PROGRAM OP90_MASTER3_IO
VAR
    OP90_MAS3_PORT1_BYTE1_DI_MODULE_1 AT %I* : BYTE;
	OP90_MAS3_PORT1_BYTE2_DI_MODULE_1 AT %I* : BYTE;
	OP90_MAS3_PORT2_BYTE1_DI_MODULE_2 AT %I* : BYTE;
	OP90_MAS3_PORT2_BYTE2_DI_MODULE_2 AT %I* : BYTE;
	OP90_MAS3_PORT3_BYTE1_DI_MODULE_3 AT %I* : BYTE;
	OP90_MAS3_PORT3_BYTE2_DI_MODULE_3 AT %I* : BYTE;
	
	OP90_MAS3_PORT5_BYTE1_DO_MODULE_1 AT %Q* : BYTE;
	OP90_MAS3_PORT5_BYTE2_DO_MODULE_1 AT %Q* : BYTE;
	OP90_MAS3_PORT5_BYTE3_DO_MODULE_1 AT %Q* : BYTE;
	OP90_MAS3_PORT6_BYTE1_DO_MODULE_2 AT %Q* : BYTE;
	OP90_MAS3_PORT6_BYTE2_DO_MODULE_2 AT %Q* : BYTE;
	OP90_MAS3_PORT7_BYTE1_DO_MODULE_3 AT %Q* : BYTE; 
	OP90_MAS3_PORT7_BYTE2_DO_MODULE_3 AT %Q* : BYTE;
	OP90_MAS3_PORT7_BYTE3_DO_MODULE_3 AT %Q* : BYTE;
	
	

	BYTE_AS_BIT_0: BYTE_AS_BIT;
	BYTE_AS_BIT_1: BYTE_AS_BIT;
	BYTE_AS_BIT_2: BYTE_AS_BIT;
	BYTE_AS_BIT_3: BYTE_AS_BIT;
	BYTE_AS_BIT_4: BYTE_AS_BIT;
	BYTE_AS_BIT_5: BYTE_AS_BIT;
	
	
	
	BIT_AS_BYTE_0: BIT_AS_BYTE;
	BIT_AS_BYTE_1: BIT_AS_BYTE;
	BIT_AS_BYTE_2: BIT_AS_BYTE;
	BIT_AS_BYTE_3: BIT_AS_BYTE;
	BIT_AS_BYTE_4: BIT_AS_BYTE;
	BIT_AS_BYTE_5: BIT_AS_BYTE;
	BIT_AS_BYTE_6: BIT_AS_BYTE;
	BIT_AS_BYTE_7: BIT_AS_BYTE;
		
END_VAR

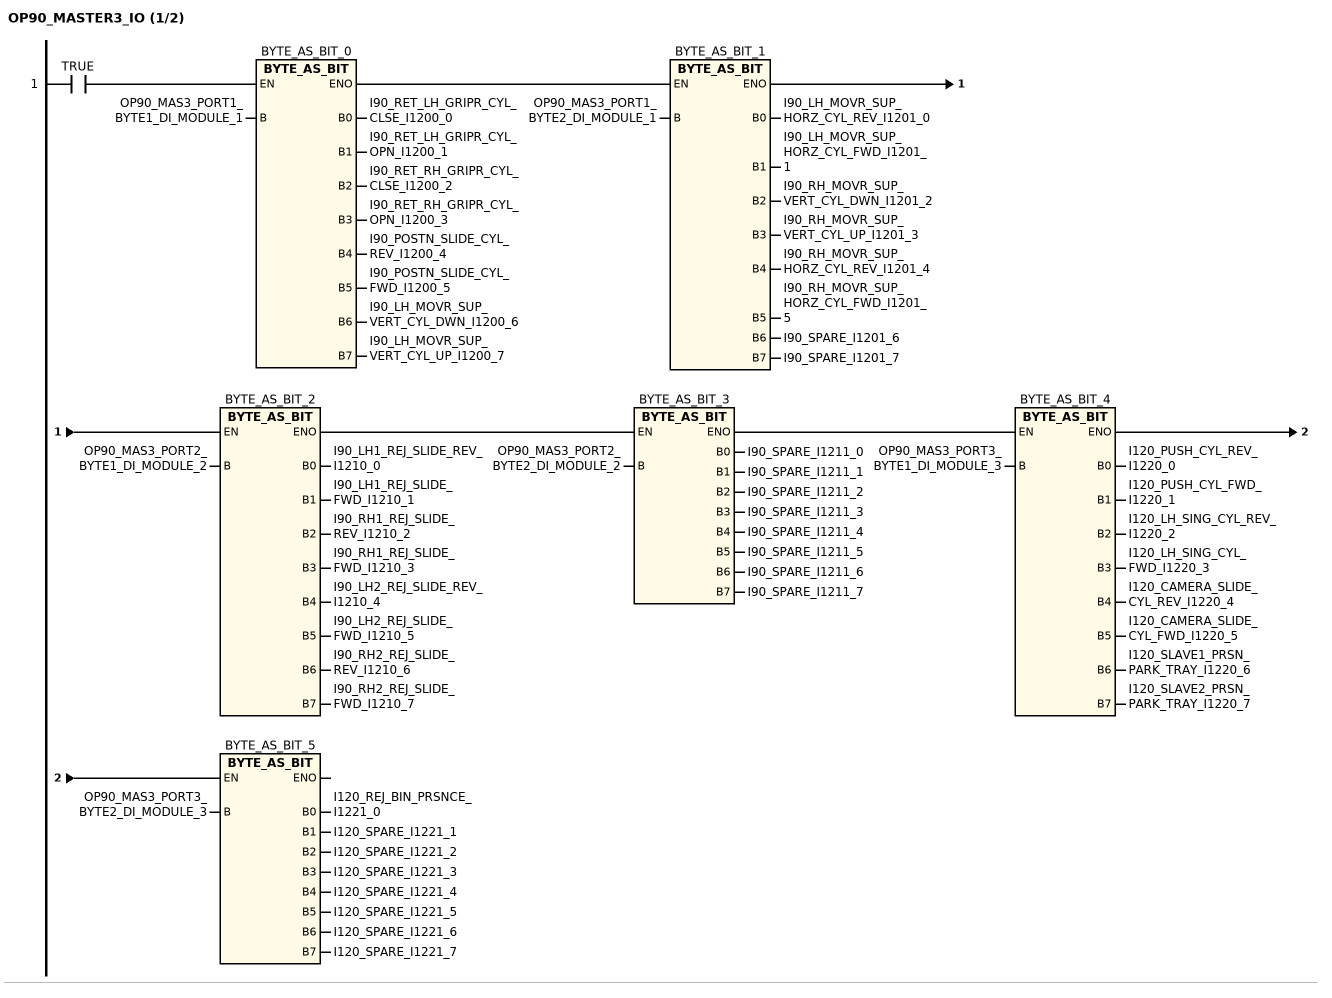
// NETWORK 1
BYTE_AS_BIT_0(
    B := OP90_MAS3_PORT1_BYTE1_DI_MODULE_1,
    B0 => I90_RET_LH_GRIPR_CYL_CLSE_I1200_0,
    B1 => I90_RET_LH_GRIPR_CYL_OPN_I1200_1,
    B2 => I90_RET_RH_GRIPR_CYL_CLSE_I1200_2,
    B3 => I90_RET_RH_GRIPR_CYL_OPN_I1200_3,
    B4 => I90_POSTN_SLIDE_CYL_REV_I1200_4,
    B5 => I90_POSTN_SLIDE_CYL_FWD_I1200_5,
    B6 => I90_LH_MOVR_SUP_VERT_CYL_DWN_I1200_6,
    B7 => I90_LH_MOVR_SUP_VERT_CYL_UP_I1200_7); // BYTE_AS_BIT
BYTE_AS_BIT_1(
    B := OP90_MAS3_PORT1_BYTE2_DI_MODULE_1,
    B0 => I90_LH_MOVR_SUP_HORZ_CYL_REV_I1201_0,
    B1 => I90_LH_MOVR_SUP_HORZ_CYL_FWD_I1201_1,
    B2 => I90_RH_MOVR_SUP_VERT_CYL_DWN_I1201_2,
    B3 => I90_RH_MOVR_SUP_VERT_CYL_UP_I1201_3,
    B4 => I90_RH_MOVR_SUP_HORZ_CYL_REV_I1201_4,
    B5 => I90_RH_MOVR_SUP_HORZ_CYL_FWD_I1201_5,
    B6 => I90_SPARE_I1201_6,
    B7 => I90_SPARE_I1201_7); // BYTE_AS_BIT
BYTE_AS_BIT_2(
    B := OP90_MAS3_PORT2_BYTE1_DI_MODULE_2,
    B0 => I90_LH1_REJ_SLIDE_REV_I1210_0,
    B1 => I90_LH1_REJ_SLIDE_FWD_I1210_1,
    B2 => I90_RH1_REJ_SLIDE_REV_I1210_2,
    B3 => I90_RH1_REJ_SLIDE_FWD_I1210_3,
    B4 => I90_LH2_REJ_SLIDE_REV_I1210_4,
    B5 => I90_LH2_REJ_SLIDE_FWD_I1210_5,
    B6 => I90_RH2_REJ_SLIDE_REV_I1210_6,
    B7 => I90_RH2_REJ_SLIDE_FWD_I1210_7); // BYTE_AS_BIT
BYTE_AS_BIT_3(
    B := OP90_MAS3_PORT2_BYTE2_DI_MODULE_2,
    B0 => I90_SPARE_I1211_0,
    B1 => I90_SPARE_I1211_1,
    B2 => I90_SPARE_I1211_2,
    B3 => I90_SPARE_I1211_3,
    B4 => I90_SPARE_I1211_4,
    B5 => I90_SPARE_I1211_5,
    B6 => I90_SPARE_I1211_6,
    B7 => I90_SPARE_I1211_7); // BYTE_AS_BIT
BYTE_AS_BIT_4(
    B := OP90_MAS3_PORT3_BYTE1_DI_MODULE_3,
    B0 => I120_PUSH_CYL_REV_I1220_0,
    B1 => I120_PUSH_CYL_FWD_I1220_1,
    B2 => I120_LH_SING_CYL_REV_I1220_2,
    B3 => I120_LH_SING_CYL_FWD_I1220_3,
    B4 => I120_CAMERA_SLIDE_CYL_REV_I1220_4,
    B5 => I120_CAMERA_SLIDE_CYL_FWD_I1220_5,
    B6 => I120_SLAVE1_PRSN_PARK_TRAY_I1220_6,
    B7 => I120_SLAVE2_PRSN_PARK_TRAY_I1220_7); // BYTE_AS_BIT
BYTE_AS_BIT_5(
    B := OP90_MAS3_PORT3_BYTE2_DI_MODULE_3,
    B0 => I120_REJ_BIN_PRSNCE_I1221_0,
    B1 => I120_SPARE_I1221_1,
    B2 => I120_SPARE_I1221_2,
    B3 => I120_SPARE_I1221_3,
    B4 => I120_SPARE_I1221_4,
    B5 => I120_SPARE_I1221_5,
    B6 => I120_SPARE_I1221_6,
    B7 => I120_SPARE_I1221_7); // BYTE_AS_BIT

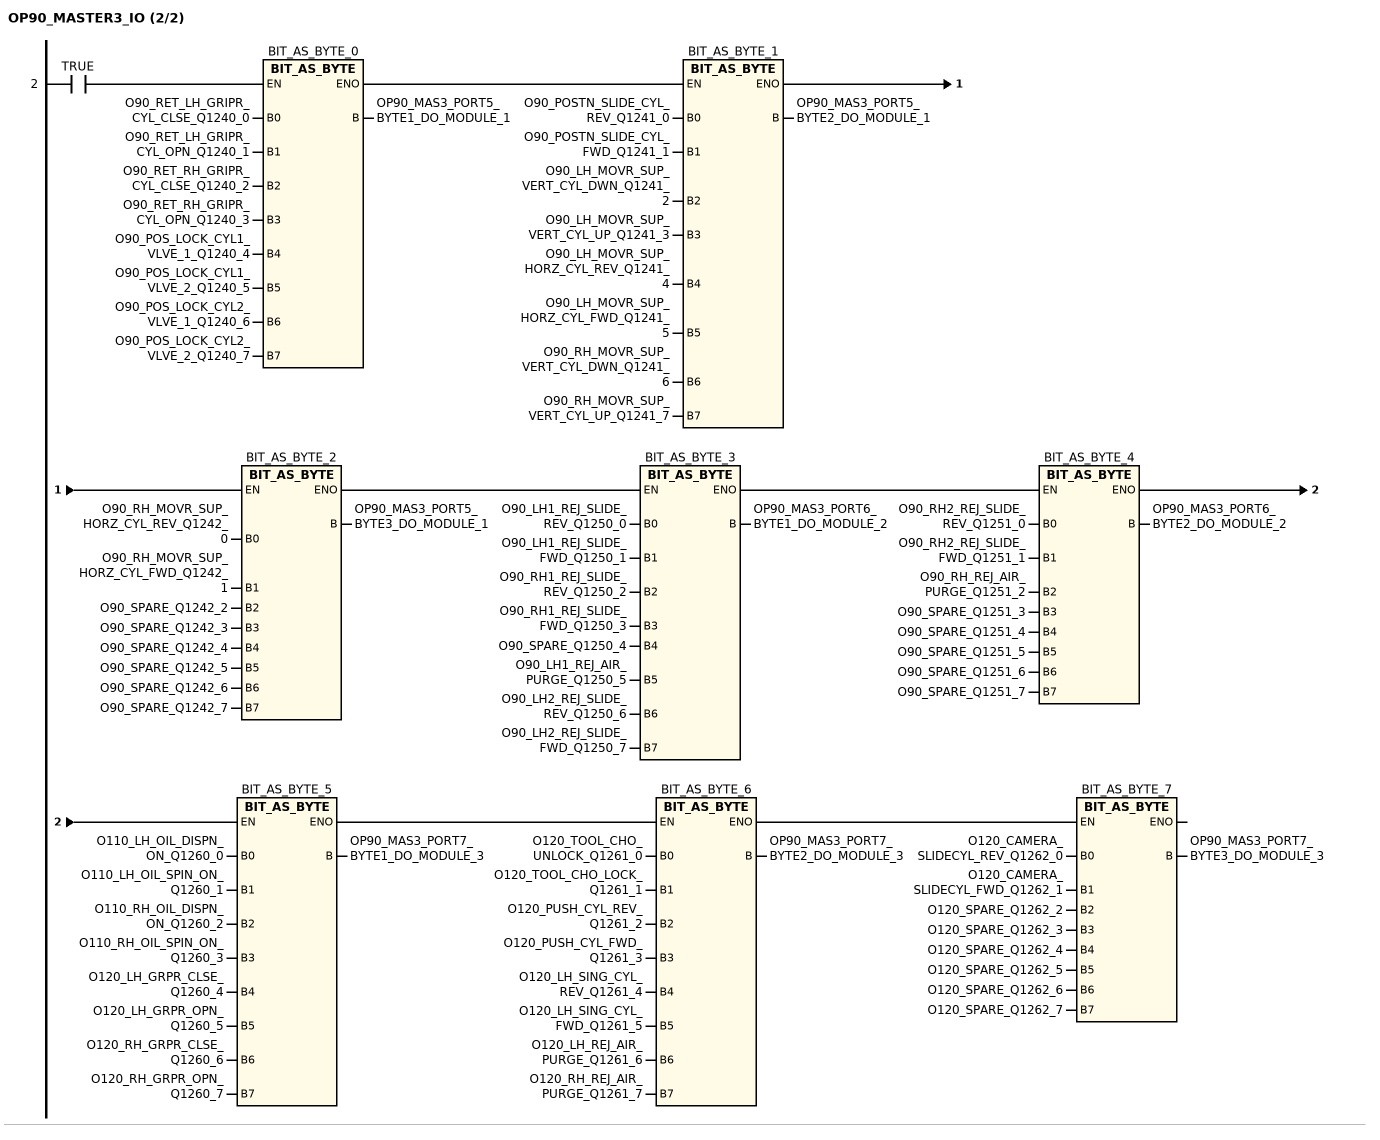
// NETWORK 2
BIT_AS_BYTE_0(
    B0 := O90_RET_LH_GRIPR_CYL_CLSE_Q1240_0,
    B1 := O90_RET_LH_GRIPR_CYL_OPN_Q1240_1,
    B2 := O90_RET_RH_GRIPR_CYL_CLSE_Q1240_2,
    B3 := O90_RET_RH_GRIPR_CYL_OPN_Q1240_3,
    B4 := O90_POS_LOCK_CYL1_VLVE_1_Q1240_4,
    B5 := O90_POS_LOCK_CYL1_VLVE_2_Q1240_5,
    B6 := O90_POS_LOCK_CYL2_VLVE_1_Q1240_6,
    B7 := O90_POS_LOCK_CYL2_VLVE_2_Q1240_7,
    B => OP90_MAS3_PORT5_BYTE1_DO_MODULE_1); // BIT_AS_BYTE
BIT_AS_BYTE_1(
    B0 := O90_POSTN_SLIDE_CYL_REV_Q1241_0,
    B1 := O90_POSTN_SLIDE_CYL_FWD_Q1241_1,
    B2 := O90_LH_MOVR_SUP_VERT_CYL_DWN_Q1241_2,
    B3 := O90_LH_MOVR_SUP_VERT_CYL_UP_Q1241_3,
    B4 := O90_LH_MOVR_SUP_HORZ_CYL_REV_Q1241_4,
    B5 := O90_LH_MOVR_SUP_HORZ_CYL_FWD_Q1241_5,
    B6 := O90_RH_MOVR_SUP_VERT_CYL_DWN_Q1241_6,
    B7 := O90_RH_MOVR_SUP_VERT_CYL_UP_Q1241_7,
    B => OP90_MAS3_PORT5_BYTE2_DO_MODULE_1); // BIT_AS_BYTE
BIT_AS_BYTE_2(
    B0 := O90_RH_MOVR_SUP_HORZ_CYL_REV_Q1242_0,
    B1 := O90_RH_MOVR_SUP_HORZ_CYL_FWD_Q1242_1,
    B2 := O90_SPARE_Q1242_2,
    B3 := O90_SPARE_Q1242_3,
    B4 := O90_SPARE_Q1242_4,
    B5 := O90_SPARE_Q1242_5,
    B6 := O90_SPARE_Q1242_6,
    B7 := O90_SPARE_Q1242_7,
    B => OP90_MAS3_PORT5_BYTE3_DO_MODULE_1); // BIT_AS_BYTE
BIT_AS_BYTE_3(
    B0 := O90_LH1_REJ_SLIDE_REV_Q1250_0,
    B1 := O90_LH1_REJ_SLIDE_FWD_Q1250_1,
    B2 := O90_RH1_REJ_SLIDE_REV_Q1250_2,
    B3 := O90_RH1_REJ_SLIDE_FWD_Q1250_3,
    B4 := O90_SPARE_Q1250_4,
    B5 := O90_LH1_REJ_AIR_PURGE_Q1250_5,
    B6 := O90_LH2_REJ_SLIDE_REV_Q1250_6,
    B7 := O90_LH2_REJ_SLIDE_FWD_Q1250_7,
    B => OP90_MAS3_PORT6_BYTE1_DO_MODULE_2); // BIT_AS_BYTE
BIT_AS_BYTE_4(
    B0 := O90_RH2_REJ_SLIDE_REV_Q1251_0,
    B1 := O90_RH2_REJ_SLIDE_FWD_Q1251_1,
    B2 := O90_RH_REJ_AIR_PURGE_Q1251_2,
    B3 := O90_SPARE_Q1251_3,
    B4 := O90_SPARE_Q1251_4,
    B5 := O90_SPARE_Q1251_5,
    B6 := O90_SPARE_Q1251_6,
    B7 := O90_SPARE_Q1251_7,
    B => OP90_MAS3_PORT6_BYTE2_DO_MODULE_2); // BIT_AS_BYTE
BIT_AS_BYTE_5(
    B0 := O110_LH_OIL_DISPN_ON_Q1260_0,
    B1 := O110_LH_OIL_SPIN_ON_Q1260_1,
    B2 := O110_RH_OIL_DISPN_ON_Q1260_2,
    B3 := O110_RH_OIL_SPIN_ON_Q1260_3,
    B4 := O120_LH_GRPR_CLSE_Q1260_4,
    B5 := O120_LH_GRPR_OPN_Q1260_5,
    B6 := O120_RH_GRPR_CLSE_Q1260_6,
    B7 := O120_RH_GRPR_OPN_Q1260_7,
    B => OP90_MAS3_PORT7_BYTE1_DO_MODULE_3); // BIT_AS_BYTE
BIT_AS_BYTE_6(
    B0 := O120_TOOL_CHO_UNLOCK_Q1261_0,
    B1 := O120_TOOL_CHO_LOCK_Q1261_1,
    B2 := O120_PUSH_CYL_REV_Q1261_2,
    B3 := O120_PUSH_CYL_FWD_Q1261_3,
    B4 := O120_LH_SING_CYL_REV_Q1261_4,
    B5 := O120_LH_SING_CYL_FWD_Q1261_5,
    B6 := O120_LH_REJ_AIR_PURGE_Q1261_6,
    B7 := O120_RH_REJ_AIR_PURGE_Q1261_7,
    B => OP90_MAS3_PORT7_BYTE2_DO_MODULE_3); // BIT_AS_BYTE
BIT_AS_BYTE_7(
    B0 := O120_CAMERA_SLIDECYL_REV_Q1262_0,
    B1 := O120_CAMERA_SLIDECYL_FWD_Q1262_1,
    B2 := O120_SPARE_Q1262_2,
    B3 := O120_SPARE_Q1262_3,
    B4 := O120_SPARE_Q1262_4,
    B5 := O120_SPARE_Q1262_5,
    B6 := O120_SPARE_Q1262_6,
    B7 := O120_SPARE_Q1262_7,
    B => OP90_MAS3_PORT7_BYTE3_DO_MODULE_3); // BIT_AS_BYTE

END_PROGRAM

(* stored: Version 1.1.0.1, ProductVersion 3.1.4024.11
   POU OP90_MASTER3_IO: Id {2c7d9cce-9354-494b-ad67-0aacc0f3c2f1}, SpecialFunc None *)
